KUKA KRL program: chk_w3_wechs_ok.src

&ACCESS RV1
&REL 4
&COMMENT Check C2
DEF chk_w3_wechs_ok( )

; VERIFICAÇÃO DE FERRAMENTA: C2

wait for (($in[161]) and ($in[169]) and (not $in[177]) and ($in[185]) and ($in[219]))


;//---- End -------
;Diag_Appl(#Off,5)
END
